ABB RAPID module: ReplayTargets_v15.mod

MODULE ReplayTargets_v15
    ! Generated from tests_v15.csv and success_v15.csv.
    ! Target names include version and testId. B* variants include version, testId, and confId.

    ! Robtargets and jointtargets for replay
    CONST robtarget rA_v15_t1 := [[1867.5,0,1823],[2.18557E-8,0,-1,0],[0,0,0,0],[9E+09,9E+09,9E+09,9E+09,9E+09,9E+09]];
    CONST robtarget rB_v15_t1 := [[1508.56,1567.66,126.218],[0.278559,-0.953814,-0.0346758,-0.10696],[0,1,1,0],[9E+09,9E+09,9E+09,9E+09,9E+09,9E+09]];
    CONST robtarget rB_v15_t1_c2 := [[1508.56,1567.66,126.218],[0.278559,-0.953814,-0.0346758,-0.10696],[0,0,-4,0],[9E+09,9E+09,9E+09,9E+09,9E+09,9E+09]];
    CONST robtarget rB_v15_t1_c5 := [[1508.56,1567.66,126.218],[0.278559,-0.953814,-0.0346758,-0.10696],[0,0,0,0],[9E+09,9E+09,9E+09,9E+09,9E+09,9E+09]];
    CONST jointtarget jA_v15_t1 := [[0,-2.3802E-6,7.25062E-7,0,90,0],[9E+09,9E+09,9E+09,9E+09,9E+09,9E+09]];
    CONST jointtarget jB_v15_t1 := [[44.9995,44.3,13.8,90.0005,14.5,134.999],[9E+09,9E+09,9E+09,9E+09,9E+09,9E+09]];
    CONST jointtarget jBseed_v15_t1 := [[45,44.3,13.8,90,14.5,135],[9E+09,9E+09,9E+09,9E+09,9E+09,9E+09]];
    CONST num seedB_v15_t1 := 7400;

    CONST robtarget rA_v15_t2 := [[1508.56,1567.66,126.218],[0.278559,-0.953814,-0.0346758,-0.10696],[0,1,1,0],[9E+09,9E+09,9E+09,9E+09,9E+09,9E+09]];
    CONST robtarget rB_v15_t2 := [[-24.9498,2276.1,2674.33],[0.285673,-0.269839,0.479571,0.784595],[0,0,-4,0],[9E+09,9E+09,9E+09,9E+09,9E+09,9E+09]];
    CONST robtarget rB_v15_t2_c8 := [[-24.9498,2276.1,2674.33],[0.285673,-0.269839,0.479571,0.784595],[0,0,4,0],[9E+09,9E+09,9E+09,9E+09,9E+09,9E+09]];
    CONST jointtarget jA_v15_t2 := [[44.9995,44.3,13.8,90.0005,14.5,134.999],[9E+09,9E+09,9E+09,9E+09,9E+09,9E+09]];
    CONST jointtarget jB_v15_t2 := [[89.9999,32.5,-64.7,45.0005,12.2,-359.999],[9E+09,9E+09,9E+09,9E+09,9E+09,9E+09]];
    CONST jointtarget jBseed_v15_t2 := [[90,32.5,-64.7,45,12.2,-360],[9E+09,9E+09,9E+09,9E+09,9E+09,9E+09]];
    CONST num seedB_v15_t2 := 15040;

    CONST robtarget rA_v15_t3 := [[-24.9498,2276.1,2674.33],[0.285673,-0.269839,0.479571,0.784595],[0,0,-4,0],[9E+09,9E+09,9E+09,9E+09,9E+09,9E+09]];
    CONST robtarget rB_v15_t3 := [[-767.321,670.136,3173.81],[0.818119,-0.240097,-0.312902,0.418482],[1,-3,-2,0],[9E+09,9E+09,9E+09,9E+09,9E+09,9E+09]];
    CONST robtarget rB_v15_t3_c2 := [[-767.321,670.136,3173.81],[0.818119,-0.240097,-0.312902,0.418482],[0,0,-4,0],[9E+09,9E+09,9E+09,9E+09,9E+09,9E+09]];
    CONST jointtarget jA_v15_t3 := [[89.9999,32.5,-64.7,45.0005,12.2,-359.999],[9E+09,9E+09,9E+09,9E+09,9E+09,9E+09]];
    CONST jointtarget jB_v15_t3 := [[135,-13.7,-35.4,-269.999,24.3,-179.999],[9E+09,9E+09,9E+09,9E+09,9E+09,9E+09]];
    CONST jointtarget jBseed_v15_t3 := [[135,-13.7,-35.4,-270,24.3,-180],[9E+09,9E+09,9E+09,9E+09,9E+09,9E+09]];
    CONST num seedB_v15_t3 := 12486;

    CONST robtarget rA_v15_t4 := [[-767.321,670.136,3173.81],[0.818119,-0.240097,-0.312902,0.418482],[1,-3,-2,0],[9E+09,9E+09,9E+09,9E+09,9E+09,9E+09]];
    CONST robtarget rB_v15_t4 := [[1907.53,-1907.5,1248.82],[0.449302,1.31724E-6,0.772179,-0.449296],[-1,-2,1,0],[9E+09,9E+09,9E+09,9E+09,9E+09,9E+09]];
    CONST robtarget rB_v15_t4_c4 := [[1907.53,-1907.5,1248.82],[0.449302,1.31724E-6,0.772179,-0.449296],[0,-4,0,0],[9E+09,9E+09,9E+09,9E+09,9E+09,9E+09]];
    CONST jointtarget jA_v15_t4 := [[135,-13.7,-35.4,-269.999,24.3,-179.999],[9E+09,9E+09,9E+09,9E+09,9E+09,9E+09]];
    CONST jointtarget jB_v15_t4 := [[-44.9997,37.3,-19.6,-179.999,6.6,135],[9E+09,9E+09,9E+09,9E+09,9E+09,9E+09]];
    CONST jointtarget jBseed_v15_t4 := [[-45,37.3,-19.6,-180,6.6,135],[9E+09,9E+09,9E+09,9E+09,9E+09,9E+09]];
    CONST num seedB_v15_t4 := 7670;

    CONST robtarget rA_v15_t5 := [[1907.53,-1907.5,1248.82],[0.449302,1.31724E-6,0.772179,-0.449296],[-1,-2,1,0],[9E+09,9E+09,9E+09,9E+09,9E+09,9E+09]];
    CONST robtarget rB_v15_t5 := [[1272.97,-1133.08,2903.66],[0.774617,-0.294771,0.130827,-0.544025],[-1,1,-2,0],[9E+09,9E+09,9E+09,9E+09,9E+09,9E+09]];
    CONST robtarget rB_v15_t5_c4 := [[1272.97,-1133.08,2903.66],[0.774617,-0.294771,0.130827,-0.544025],[0,-4,0,0],[9E+09,9E+09,9E+09,9E+09,9E+09,9E+09]];
    CONST jointtarget jA_v15_t5 := [[-44.9997,37.3,-19.6,-179.999,6.6,135],[9E+09,9E+09,9E+09,9E+09,9E+09,9E+09]];
    CONST jointtarget jB_v15_t5 := [[-45.0003,7.8,-39.9,134.999,56.9,-179.999],[9E+09,9E+09,9E+09,9E+09,9E+09,9E+09]];
    CONST jointtarget jBseed_v15_t5 := [[-45,7.8,-39.9,135,56.9,-180],[9E+09,9E+09,9E+09,9E+09,9E+09,9E+09]];
    CONST num seedB_v15_t5 := 10027;

    CONST robtarget rA_v15_t6 := [[1272.97,-1133.08,2903.66],[0.774617,-0.294771,0.130827,-0.544025],[-1,1,-2,0],[9E+09,9E+09,9E+09,9E+09,9E+09,9E+09]];
    CONST robtarget rB_v15_t6 := [[-103.495,-2417.03,602.331],[0.125073,-0.454861,-0.741281,0.477452],[-1,3,0,0],[9E+09,9E+09,9E+09,9E+09,9E+09,9E+09]];
    CONST robtarget rB_v15_t6_c3 := [[-103.495,-2417.03,602.331],[0.125073,-0.454861,-0.741281,0.477452],[0,4,-4,0],[9E+09,9E+09,9E+09,9E+09,9E+09,9E+09]];
    CONST jointtarget jA_v15_t6 := [[-45.0003,7.8,-39.9,134.999,56.9,-179.999],[9E+09,9E+09,9E+09,9E+09,9E+09,9E+09]];
    CONST jointtarget jB_v15_t6 := [[-89.9998,38.4,2.4,270,38.3,45.0002],[9E+09,9E+09,9E+09,9E+09,9E+09,9E+09]];
    CONST jointtarget jBseed_v15_t6 := [[-90,38.4,2.4,270,38.3,45],[9E+09,9E+09,9E+09,9E+09,9E+09,9E+09]];
    CONST num seedB_v15_t6 := 17546;

ENDMODULE
